// TIA Portal V19 export
ORGANIZATION_BLOCK "Main"   // OB1, LAD, ProgramCycle
TITLE = "Main Program Sweep (Cycle)"
{ S7_Optimized_Access := 'TRUE' }
// stored: AutoNumber false, SetENOAutomatically false
BEGIN

REGION Network 1: Buffer inputs to send to 1500
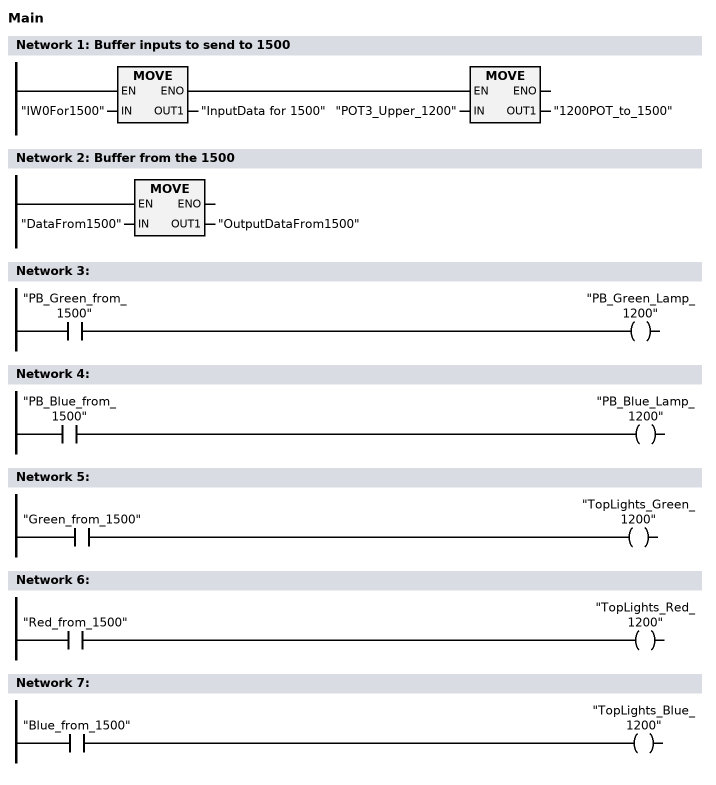
   RUNG wire#powerrail
      { S7_GenerateENO := "TRUE" } Move(in := "IW0For1500", out1 => "InputData for 1500")
      { S7_GenerateENO := "TRUE" } Move(in := "POT3_Upper_1200", out1 => "1200POT_to_1500")
   END_RUNG
   // the same network as SCL:
   // ENO of a box is taken as its EN; it also drops when the box reports an error
   "InputData for 1500" := "IW0For1500";
   "1200POT_to_1500" := "POT3_Upper_1200";
END_REGION

REGION Network 2: Buffer from the 1500
   RUNG wire#powerrail
      { S7_GenerateENO := "TRUE" } Move(in := "DataFrom1500", out1 => "OutputDataFrom1500")
   END_RUNG
   // the same network as SCL:
   "OutputDataFrom1500" := "DataFrom1500";
END_REGION

REGION Network 3
   RUNG wire#powerrail
      Contact( "PB_Green_from_1500" )
      Coil( "PB_Green_Lamp_1200" )
   END_RUNG
   // the same network as SCL:
   "PB_Green_Lamp_1200" := "PB_Green_from_1500";
END_REGION

REGION Network 4
   RUNG wire#powerrail
      Contact( "PB_Blue_from_1500" )
      Coil( "PB_Blue_Lamp_1200" )
   END_RUNG
   // the same network as SCL:
   "PB_Blue_Lamp_1200" := "PB_Blue_from_1500";
END_REGION

REGION Network 5
   RUNG wire#powerrail
      Contact( "Green_from_1500" )
      Coil( "TopLights_Green_1200" )
   END_RUNG
   // the same network as SCL:
   "TopLights_Green_1200" := "Green_from_1500";
END_REGION

REGION Network 6
   RUNG wire#powerrail
      Contact( "Red_from_1500" )
      Coil( "TopLights_Red_1200" )
   END_RUNG
   // the same network as SCL:
   "TopLights_Red_1200" := "Red_from_1500";
END_REGION

REGION Network 7
   RUNG wire#powerrail
      Contact( "Blue_from_1500" )
      Coil( "TopLights_Blue_1200" )
   END_RUNG
   // the same network as SCL:
   "TopLights_Blue_1200" := "Blue_from_1500";
END_REGION
END_ORGANIZATION_BLOCK
